# EPICS substitutions: db/MonoDAQ/ecmcMonoDAQ-E-gMeter.substitutions
file "ecmc_analogInput-chX.template"{
  pattern {CH_ID, KEY,      sourceName, ESLO, EGU,  PREC}
          {01,    counter,  counter,    1,    "",   0   }
}

file "ecmc_analogInputFloat-chX.template"{
  pattern {CH_ID, KEY,          sourceName,     ESLO, EGU,    PREC}
          {01,    temperature,  temperature,    1,    "degC", 3   }
          {01,    X,            accelerometer,  1,    "g",    6   }
          {02,    Y,            accelerometer,  1,    "g",    6   }
          {03,    Z,            accelerometer,  1,    "g",    6   }
}
